// Mitsubishi GX Works2 project: 31-4   PLC: FX3G

// global labels: Global1
VAR_GLOBAL
  start_day AT X007 : BOOL;
  YYYY AT Y007 : BOOL;
  Y1coil AT Y007 : BOOL;
  Reg_WhippedCream AT D1100 : REAL;
END_VAR
VAR_GLOBAL CONSTANT
  constant1_Inventory : REAL := 300;
END_VAR
VAR_GLOBAL
  M_InventoryWhippedCream AT M20 : BOOL;
  Reg_Biscwit AT D1102 : REAL;
END_VAR
VAR_GLOBAL CONSTANT
  constant2_Inventory : REAL := 6;
END_VAR
VAR_GLOBAL
  M_InventoryBiscwit AT Y007 : BOOL;
  Reg_Chochlet AT D1104 : REAL;
END_VAR
VAR_GLOBAL CONSTANT
  constant3_Inventory : REAL := 300;
END_VAR
VAR_GLOBAL
  M_InventoryChochlet AT Y007 : BOOL;
  M_InvetoryWhippedCream AT M20 : BOOL;
  M_InvetoryBiscwit AT M21 : BOOL;
  M_InvetoryChochlet AT M22 : BOOL;
  M_canStartDay AT M0 : BOOL;
  M_toStart AT M1 : BOOL;
  M_InvetoryWhippedCream1 AT M20 : BOOL;
  M_InvetoryBiscwit1 AT M21 : BOOL;
  M_InvetoryChochlet1 AT M22 : BOOL;
  TEXT AT Y011 : BOOL;
  TC_CloseDayTimer_3 AT TC3 : BOOL;
END_VAR
VAR_GLOBAL CONSTANT
  CONSTANT30_word : INT := 30;
END_VAR
VAR_GLOBAL
  lamp1 AT TS1 : BOOL;
  M_stoptDay AT M0 : BOOL;
  tozilof AT X011 : BOOL;
  M_foundMinimum AT X011 : BOOL;
  X011ToStart AT X011 : BOOL;
END_VAR
VAR_GLOBAL CONSTANT
  REG_MinimumCream : REAL := 300;
END_VAR
VAR_GLOBAL
  Reg_sprinkling AT D1106 : REAL;
  M007t AT M7 : BOOL;
  check7 AT M7 : BOOL;
END_VAR
VAR_GLOBAL CONSTANT
  constant1_WhippedCream : REAL := 300;
  constant_WhippedCream : REAL := 300;
  constant_Biscwit : REAL := 6;
  constant_Chochlet : REAL := 240;
  T300Cream : REAL := 300;
  CONSTANT0_float : REAL := 700;
  CONSTANT_CHOCHOLET : REAL := 500;
  CONSTANT_WP : REAL := 300;
  CONSTANT_CH : REAL := 500;
  CONSTANT_BI : REAL := 100;
END_VAR
VAR_GLOBAL
  Reset_Inventory AT M2 : BOOL;
  lamp0 AT M3 : BOOL;
  lamp00 AT M3 : BOOL;
  light0 AT M81 : BOOL;
  light1 AT M82 : BOOL;
  lamp01 AT M3 : BOOL;
END_VAR
VAR_GLOBAL CONSTANT
  TV20 : INT := 5;
END_VAR
VAR_GLOBAL
  TC_light_1 AT TC1 : BOOL;
  TS_light_0 AT TS0 : BOOL;
  TC_light_0 AT TC0 : BOOL;
  TS_light_1 AT TS1 : BOOL;
  start_dipping AT X006 : BOOL;
  SW_AnalogInput1 AT D8280 : INT;
  M_dipping AT M4 : BOOL;
END_VAR
VAR_GLOBAL CONSTANT
  CONSTANT382_1inanalog : INT := 382;
END_VAR
VAR_GLOBAL
  M_CheckDipping AT M5 : BOOL;
END_VAR
VAR_GLOBAL CONSTANT
  CONSTANT2020_5inanalog : INT := 2020;
END_VAR
VAR_GLOBAL
  M_CheckDipping5 AT M6 : BOOL;
  M_CheckDipping1 AT M5 : BOOL;
  lamp3 AT M8 : BOOL;
  SenTouch AT X001 : BOOL;
  Camera AT X002 : BOOL;
  EmergencyButton AT X005 : BOOL;
  SenTemp30 AT X003 : BOOL;
  SenTemp15 AT X004 : BOOL;
  OpenSprinkling AT M33 : BOOL;
  StartSprinkling AT X010 : BOOL;
  OpenSprinkling1 AT M6 : BOOL;
  SprinklingIsOpen AT Y004 : BOOL;
END_VAR
VAR_GLOBAL CONSTANT
  CONSTANT0_1inanalog : INT;
  CONSTANT1995_5inanalog : INT := 1995;
  CONSTANT0_0inanalog : INT;
  CONSTANT3999_10inanalog : INT := 3999;
END_VAR
VAR_GLOBAL
  M_CheckDipping2 AT M55 : BOOL;
END_VAR
VAR_GLOBAL CONSTANT
  CONSTANT2389_6inanalog : INT := 2389;
END_VAR
VAR_GLOBAL
  M_CheckDipping3 AT M66 : BOOL;
END_VAR
VAR_GLOBAL CONSTANT
  CONSTANT_CHOCHOLET20 : REAL := 120;
  CONSTANT_CHOCHOLET40 : REAL := 240;
END_VAR
VAR_GLOBAL
  YY00 AT Y000 : BOOL;
  YY11 AT Y001 : BOOL;
  Reg_dippingToDelte AT D1110 : INT;
  Reg_dipping AT D1112 : REAL;
  Dipping20On AT M11 : BOOL;
  Dipping40On AT M12 : BOOL;
  TC4 AT TC4 : BOOL;
  TC_QA_TEST_PASSED AT TC4 : BOOL;
  TC_4 AT TC4 : BOOL;
END_VAR
VAR_GLOBAL CONSTANT
  CONSTANT50 : INT := 50;
END_VAR
VAR_GLOBAL
  TS_4 AT TS4 : BOOL;
  y_3 AT Y003 : BOOL;
END_VAR
VAR_GLOBAL CONSTANT
  CONSTANT500 : INT := 50;
END_VAR
VAR_GLOBAL
  Start_packing AT X000 : BOOL;
END_VAR
VAR_GLOBAL CONSTANT
  Constant5 : INT := 5;
END_VAR
VAR_GLOBAL
  CC_Start_Squeeze_0 AT CC0 : BOOL;
  CC_counting_0 AT CC0 : BOOL;
  CS0_COUNTING AT CS0 : BOOL;
  Y2_ON AT Y002 : BOOL;
END_VAR
VAR_GLOBAL CONSTANT
  Constant6 : INT := 6;
END_VAR
VAR_GLOBAL
  CS1_COUNTING AT CS1 : BOOL;
  CC_counting_1 AT CC1 : BOOL;
END_VAR
VAR_GLOBAL CONSTANT
  CONSTANT_1 : REAL := 6;
  CONSTANT_6 : REAL := 6;
END_VAR
VAR_GLOBAL
  addto8282 AT D8282 : INT;
END_VAR
VAR_GLOBAL CONSTANT
  CONSTANT_10 : REAL := 10;
END_VAR
VAR_GLOBAL
  CS_counting_0 AT CS0 : BOOL;
  CS_counting_1 AT CS1 : BOOL;
  check_sprinkling AT M77 : BOOL;
  TC_total AT TC4 : BOOL;
END_VAR
VAR_GLOBAL CONSTANT
  TV40 : INT := 40;
END_VAR
VAR_GLOBAL
  M_300 AT M300 : BOOL;
  TS_total AT TS4 : BOOL;
  Ymove0 AT Y000 : BOOL;
  Ymove1 AT Y001 : BOOL;
  Step1 AT M101 : BOOL;
  Step2 AT M102 : BOOL;
  Step3 AT M103 : BOOL;
  Step4 AT M104 : BOOL;
  StepFinal AT M100 : BOOL;
  TC_5 AT TC5 : BOOL;
  TS_5 AT TS5 : BOOL;
  ToStep2 AT M102 : BOOL;
  TS_CloseDayTimer_3 AT TS3 : BOOL;
  Ym11 AT Y011 : BOOL;
  Step4M AT M444 : BOOL;
  Step5 AT M105 : BOOL;
  Step3M AT M333 : BOOL;
  Reg_Count_to8282 AT D1116 : INT;
  Reg_Countt AT D1122 : REAL;
  mtototot99 AT M99 : BOOL;
  Reg_Countt10 AT D1124 : REAL;
END_VAR
VAR_GLOBAL CONSTANT
  COcococo23 : INT := 2;
  CON400 : INT := 400;
  CON40 : REAL := 40;
END_VAR
VAR_GLOBAL
  Dippingn AT M11 : BOOL;
  goagain AT M110 : BOOL;
  X_11 AT Y011 : BOOL;
  Reg_fill_WP AT D1130 : REAL;
  Reg_fill_CH AT D1132 : REAL;
  Reg_fill_BI AT D1134 : REAL;
  M_reset AT M64 : BOOL;
  M_step1 AT M63 : BOOL;
END_VAR

// task Task_01 (event TRUE, interval 0, priority 31): POU_01

PROGRAM POU_01
(* structured ladder/FBD written out as ST: instructions are called as NAME(EN, inputs, outputs); _pN, _eN, _tN stand for wires *)
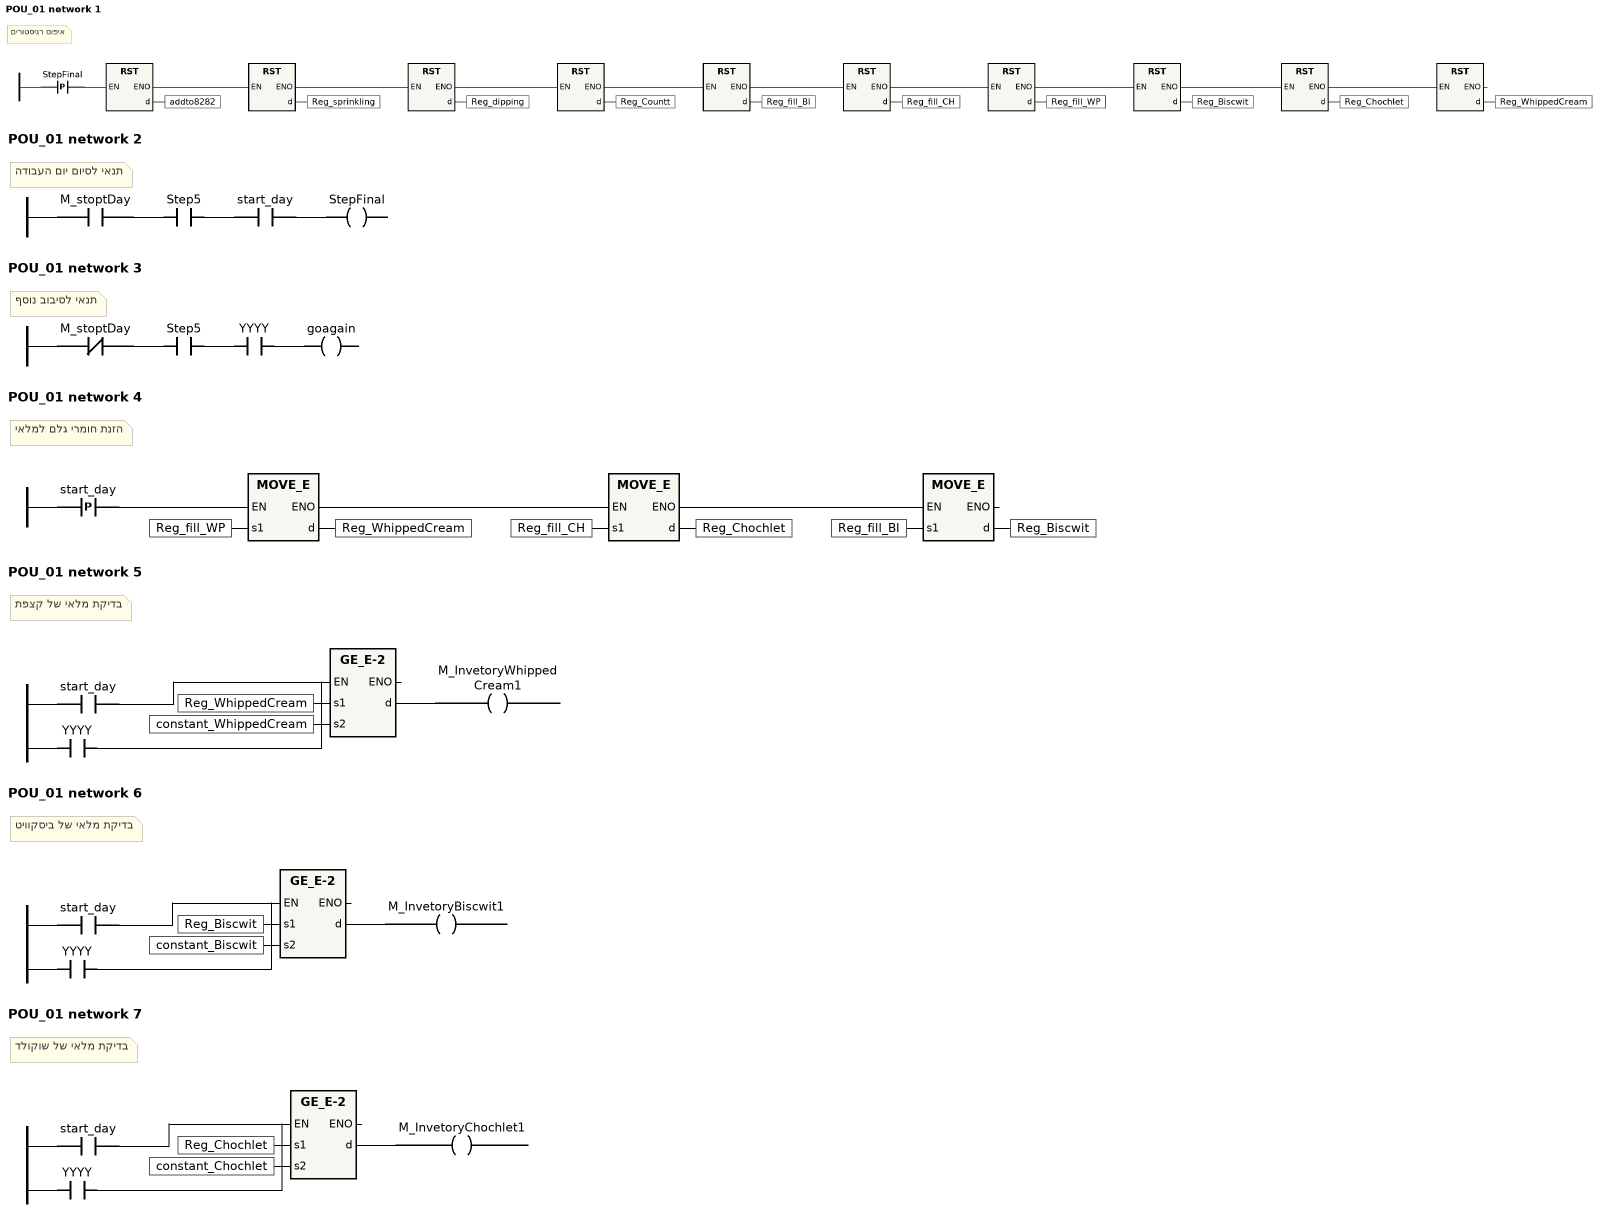
(* network 1 *)
(* איפוס רגיסטורים *)
_e1 := RST(LDP(TRUE, StepFinal), addto8282);
_e2 := RST(_e1, Reg_sprinkling);
_e3 := RST(_e2, Reg_dipping);
_e4 := RST(_e3, Reg_Countt);
_e5 := RST(_e4, Reg_fill_BI);
_e6 := RST(_e5, Reg_fill_CH);
_e7 := RST(_e6, Reg_fill_WP);
_e8 := RST(_e7, Reg_Biscwit);
_e9 := RST(_e8, Reg_Chochlet);
RST(_e9, Reg_WhippedCream);
(* network 2 *)
(* תנאי לסיום יום העבודה *)
StepFinal := M_stoptDay AND Step5 AND start_day;
(* network 3 *)
(* תנאי לסיבוב נוסף *)
goagain := NOT M_stoptDay AND Step5 AND YYYY;
(* network 4 *)
(* הזנת חומרי גלם למלאי *)
_e1 := MOVE_E(LDP(TRUE, start_day), Reg_fill_WP, Reg_WhippedCream);
_e2 := MOVE_E(_e1, Reg_fill_CH, Reg_Chochlet);
MOVE_E(_e2, Reg_fill_BI, Reg_Biscwit);
(* network 5 *)
(* בדיקת מלאי של קצפת *)
GE_E(start_day OR YYYY, Reg_WhippedCream, constant_WhippedCream, _t1);
M_InvetoryWhippedCream1 := _t1;
(* network 6 *)
(* בדיקת מלאי של ביסקוויט *)
GE_E(start_day OR YYYY, Reg_Biscwit, constant_Biscwit, _t1);
M_InvetoryBiscwit1 := _t1;
(* network 7 *)
(* בדיקת מלאי של שוקולד *)
GE_E(start_day OR YYYY, Reg_Chochlet, constant_Chochlet, _t1);
M_InvetoryChochlet1 := _t1;
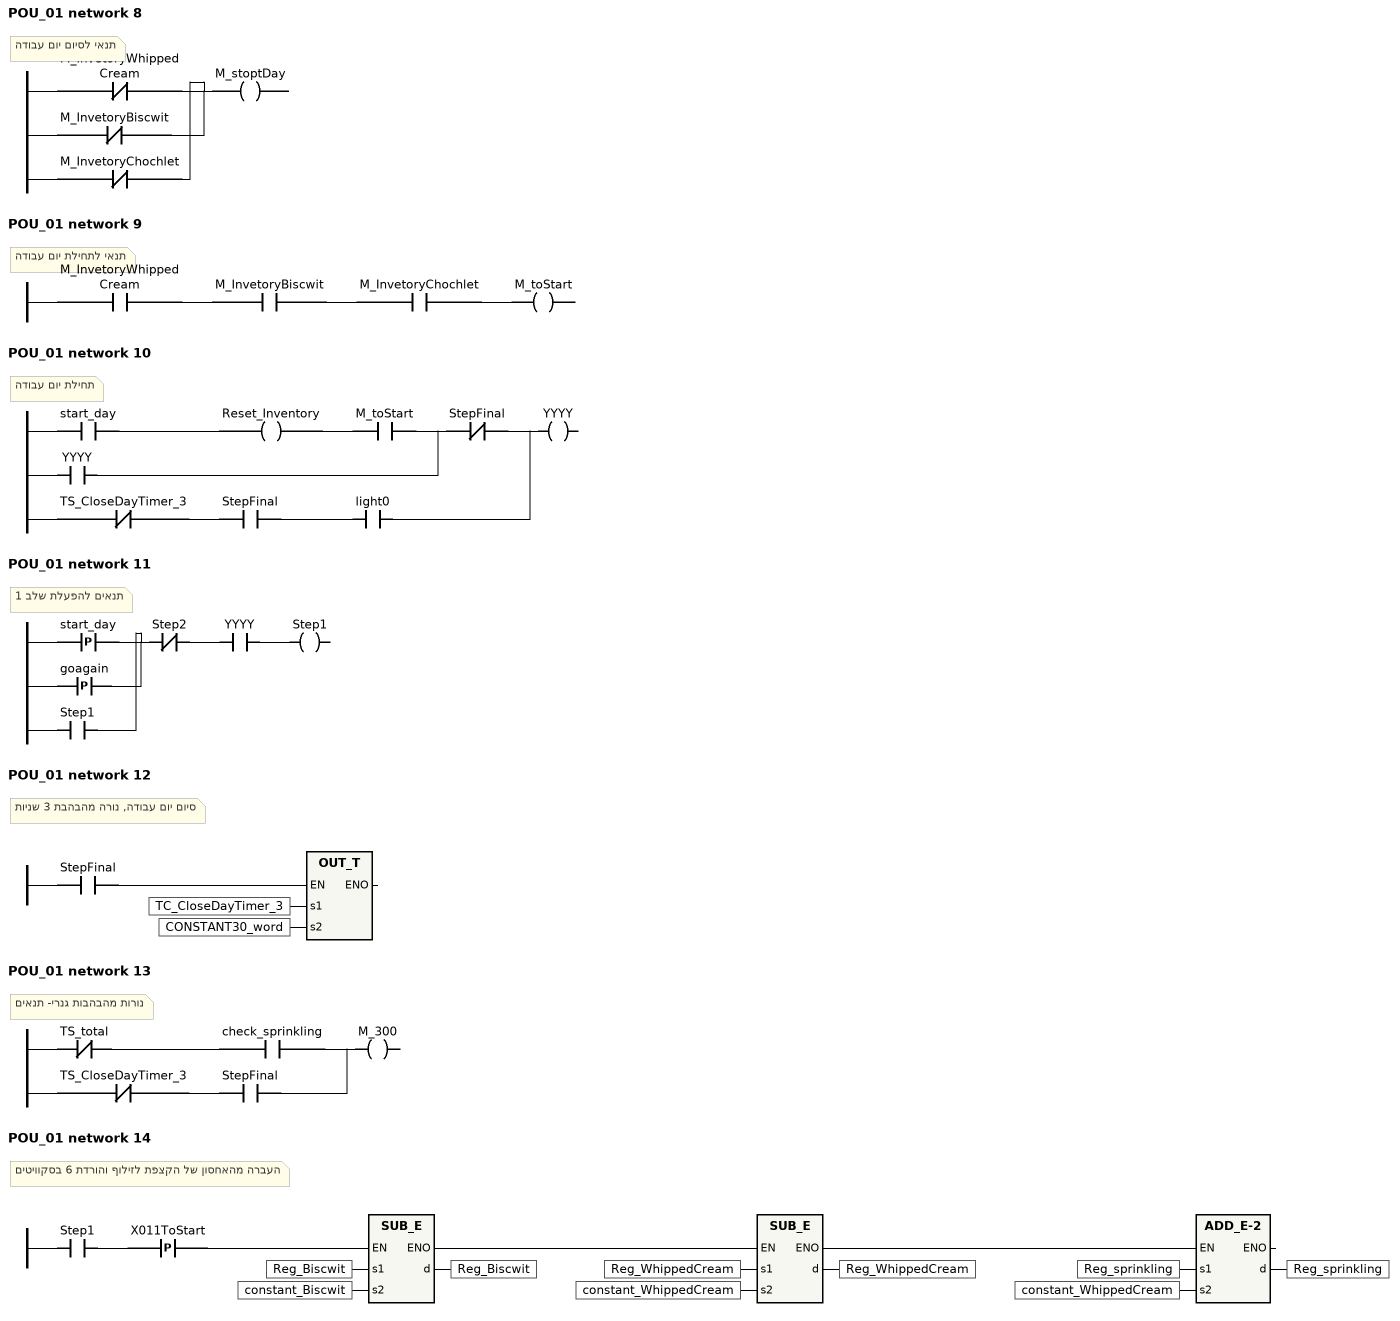
(* network 8 *)
(* תנאי לסיום יום עבודה *)
M_stoptDay := (NOT M_InvetoryWhippedCream) OR (NOT M_InvetoryBiscwit) OR (NOT M_InvetoryChochlet);
(* network 9 *)
(* תנאי לתחילת יום עבודה *)
M_toStart := M_InvetoryWhippedCream AND M_InvetoryBiscwit AND M_InvetoryChochlet;
(* network 10 *)
(* תחילת יום עבודה *)
Reset_Inventory := start_day;
YYYY := (((start_day AND M_toStart) OR YYYY) AND NOT StepFinal) OR (NOT TS_CloseDayTimer_3 AND StepFinal AND light0);
(* network 11 *)
(* תנאים להפעלת שלב 1 *)
Step1 := ((LDP(TRUE, start_day) OR LDP(TRUE, goagain) OR Step1) AND NOT Step2) AND YYYY;
(* network 12 *)
(* סיום יום עבודה, נורה מהבהבת 3 שניות *)
OUT_T(StepFinal, TC_CloseDayTimer_3, CONSTANT30_word);
(* network 13 *)
(* נורות מהבהבות גנרי- תנאים *)
M_300 := (NOT TS_total AND check_sprinkling) OR (NOT TS_CloseDayTimer_3 AND StepFinal);
(* network 14 *)
(* העברה מהאחסון של הקצפת לזילוף והורדת 6 בסקוויטים *)
_e1 := SUB_E(Step1 AND LDP(TRUE, X011ToStart), Reg_Biscwit, constant_Biscwit, Reg_Biscwit);
_e2 := SUB_E(_e1, Reg_WhippedCream, constant_WhippedCream, Reg_WhippedCream);
ADD_E(_e2, Reg_sprinkling, constant_WhippedCream, Reg_sprinkling);
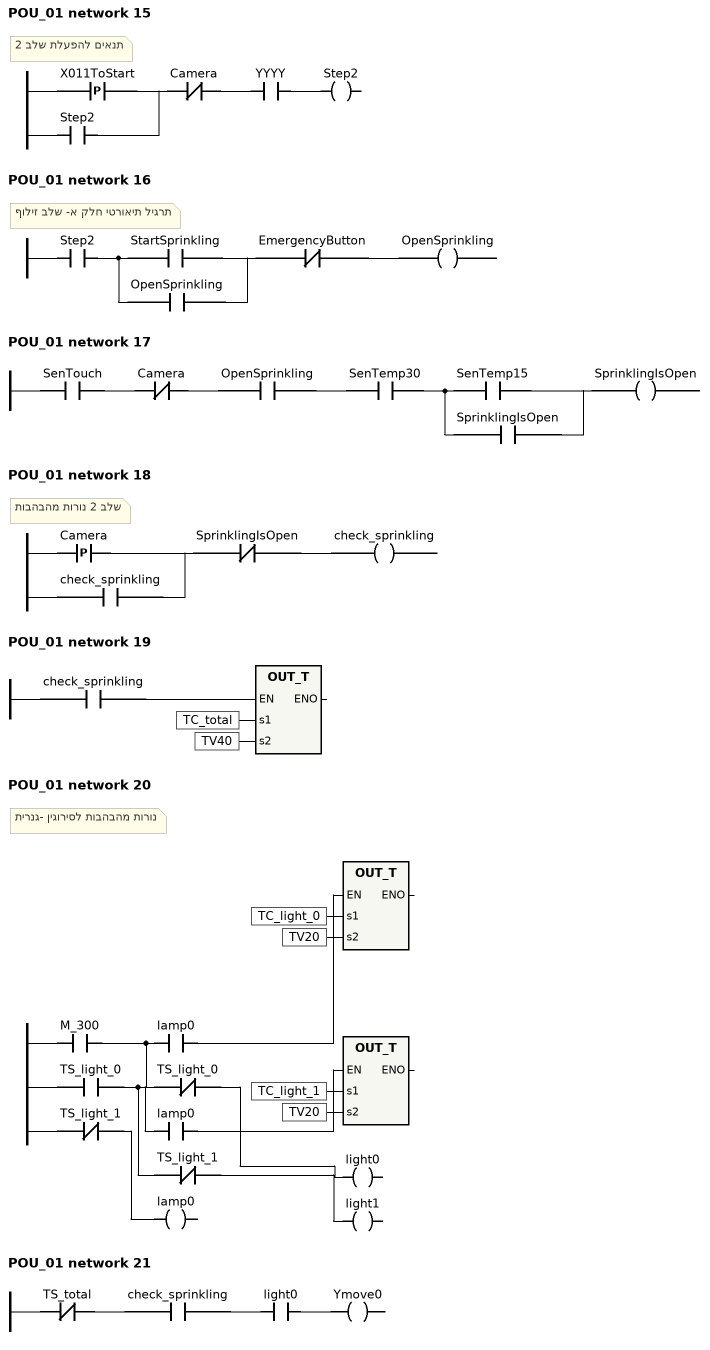
(* network 15 *)
(* תנאים להפעלת שלב 2 *)
Step2 := ((LDP(TRUE, X011ToStart) OR Step2) AND NOT Camera) AND YYYY;
(* network 16 *)
(* תרגיל תיאורטי חלק א- שלב זילוף *)
OpenSprinkling := ((Step2 AND StartSprinkling) OR (Step2 AND OpenSprinkling)) AND NOT EmergencyButton;
(* network 17 *)
_p1 := SenTouch AND NOT Camera AND OpenSprinkling AND SenTemp30;
SprinklingIsOpen := (_p1 AND SenTemp15) OR (_p1 AND SprinklingIsOpen);
(* network 18 *)
(* שלב 2 נורות מהבהבות *)
check_sprinkling := (LDP(TRUE, Camera) OR check_sprinkling) AND NOT SprinklingIsOpen;
(* network 19 *)
OUT_T(check_sprinkling, TC_total, TV40);
(* network 20 *)
(* נורות מהבהבות לסירוגין -גנרית *)
OUT_T(M_300 AND lamp0, TC_light_0, TV20);
light0 := M_300 AND NOT TS_light_0;
OUT_T(TS_light_0 AND lamp0, TC_light_1, TV20);
light1 := TS_light_0 AND NOT TS_light_1;
lamp0 := NOT TS_light_1;
(* network 21 *)
Ymove0 := NOT TS_total AND check_sprinkling AND light0;
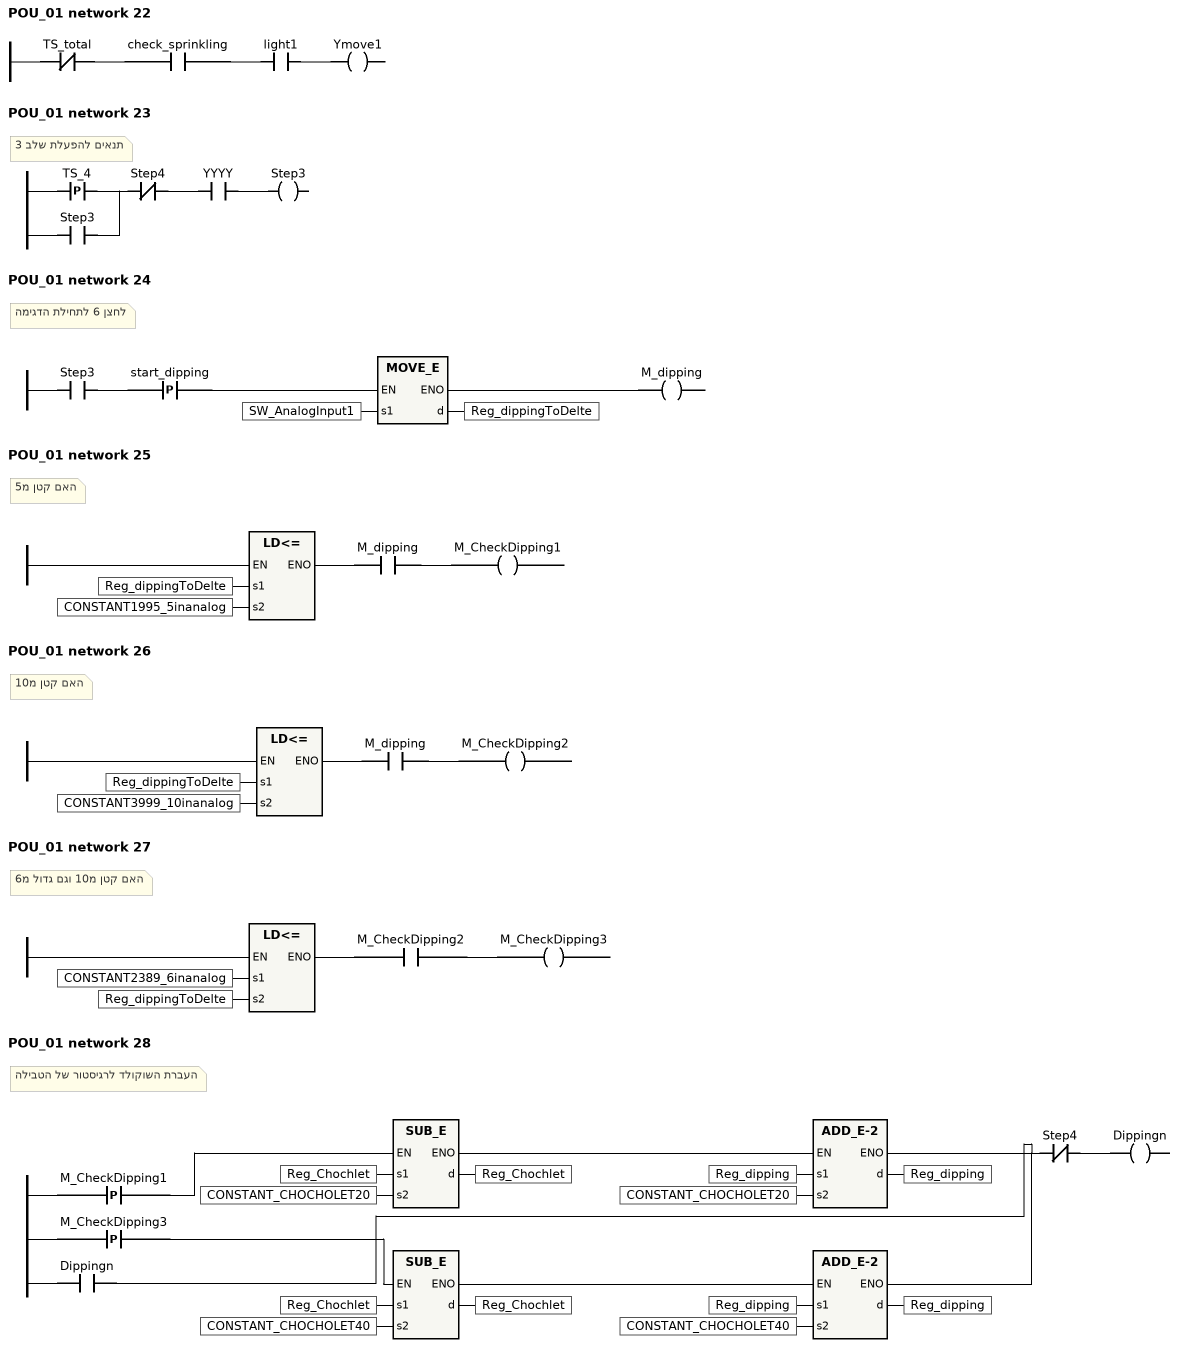
(* network 22 *)
Ymove1 := NOT TS_total AND check_sprinkling AND light1;
(* network 23 *)
(* תנאים להפעלת שלב 3 *)
Step3 := ((LDP(TRUE, TS_4) OR Step3) AND NOT Step4) AND YYYY;
(* network 24 *)
(* לחצן 6 לתחילת הדגימה *)
_e1 := MOVE_E(Step3 AND LDP(TRUE, start_dipping), SW_AnalogInput1, Reg_dippingToDelte);
M_dipping := _e1;
(* network 25 *)
(* האם קטן מ5 *)
_e1 := LD<=(TRUE, Reg_dippingToDelte, CONSTANT1995_5inanalog);
M_CheckDipping1 := _e1 AND M_dipping;
(* network 26 *)
(* האם קטן מ10 *)
_e1 := LD<=(TRUE, Reg_dippingToDelte, CONSTANT3999_10inanalog);
M_CheckDipping2 := _e1 AND M_dipping;
(* network 27 *)
(* האם קטן מ10 וגם גדול מ6 *)
_e1 := LD<=(TRUE, CONSTANT2389_6inanalog, Reg_dippingToDelte);
M_CheckDipping3 := _e1 AND M_CheckDipping2;
(* network 28 *)
(* העברת השוקולד לרגיסטור של הטבילה *)
_e1 := SUB_E(LDP(TRUE, M_CheckDipping1), Reg_Chochlet, CONSTANT_CHOCHOLET20, Reg_Chochlet);
_e2 := ADD_E(_e1, Reg_dipping, CONSTANT_CHOCHOLET20, Reg_dipping);
_e3 := SUB_E(LDP(TRUE, M_CheckDipping3), Reg_Chochlet, CONSTANT_CHOCHOLET40, Reg_Chochlet);
_e4 := ADD_E(_e3, Reg_dipping, CONSTANT_CHOCHOLET40, Reg_dipping);
Dippingn := (_e2 OR _e4 OR Dippingn) AND NOT Step4;
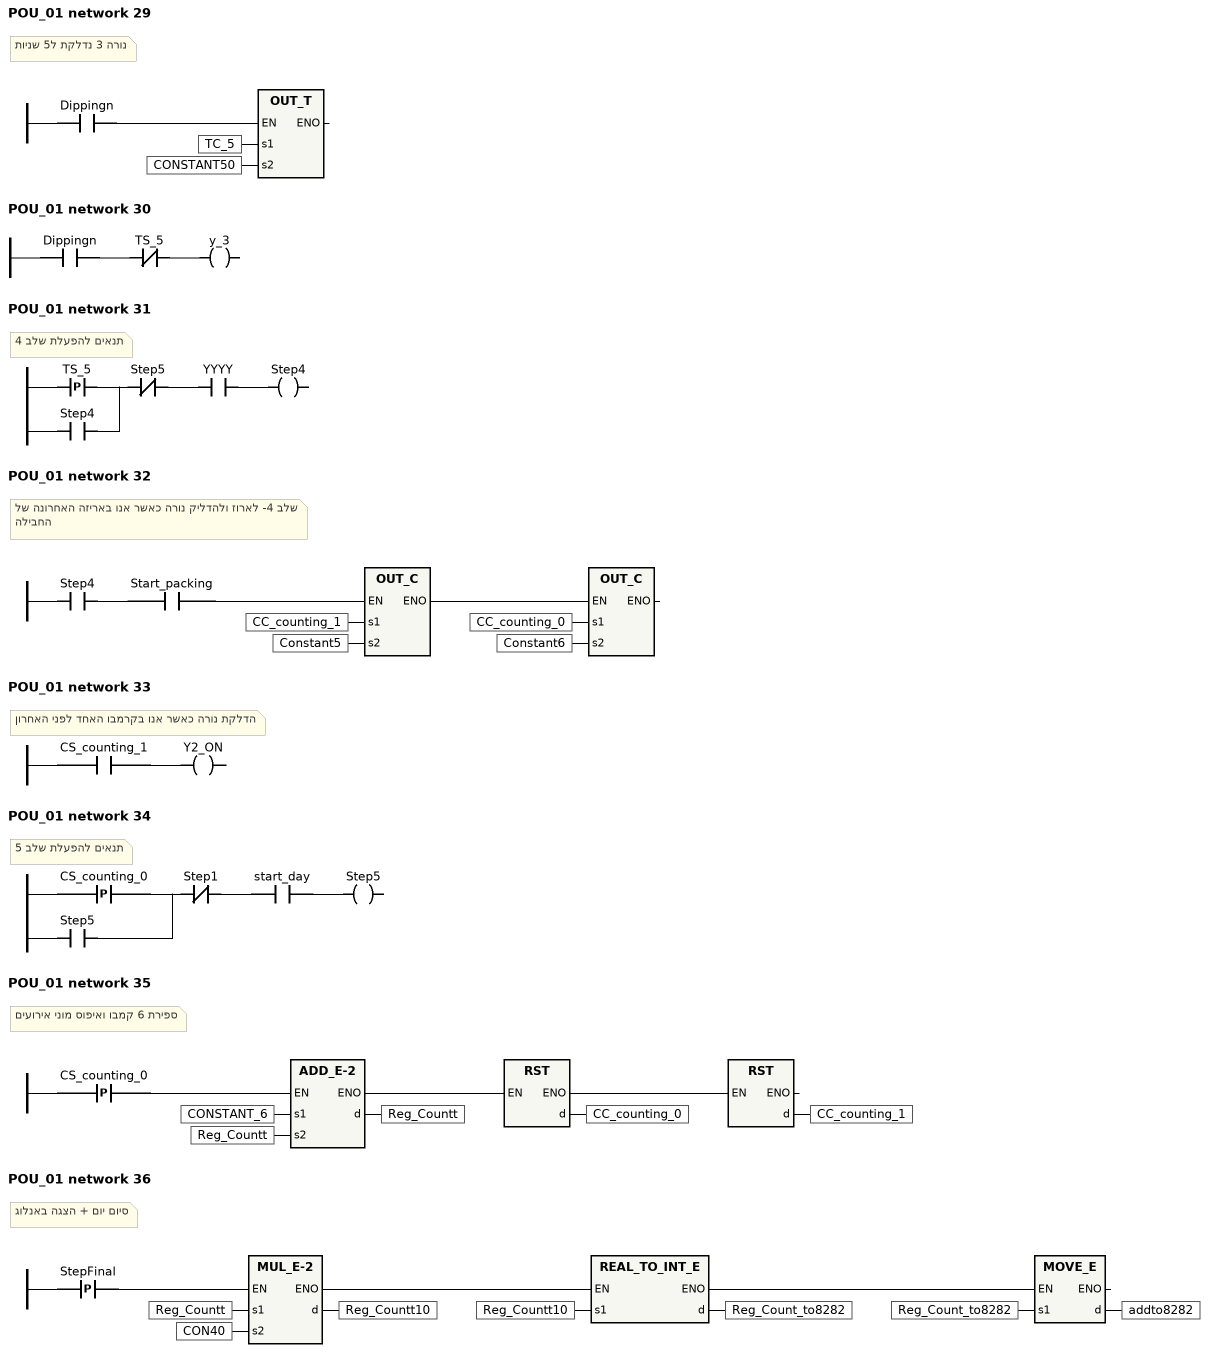
(* network 29 *)
(* נורה 3 נדלקת ל5 שניות *)
OUT_T(Dippingn, TC_5, CONSTANT50);
(* network 30 *)
y_3 := Dippingn AND NOT TS_5;
(* network 31 *)
(* תנאים להפעלת שלב 4 *)
Step4 := ((LDP(TRUE, TS_5) OR Step4) AND NOT Step5) AND YYYY;
(* network 32 *)
(* שלב 4- לארוז ולהדליק נורה כאשר אנו באריזה האחרונה של החבילה *)
_e1 := OUT_C(Step4 AND Start_packing, CC_counting_1, Constant5);
OUT_C(_e1, CC_counting_0, Constant6);
(* network 33 *)
(* הדלקת נורה כאשר אנו בקרמבו האחד לפני האחרון *)
Y2_ON := CS_counting_1;
(* network 34 *)
(* תנאים להפעלת שלב 5 *)
Step5 := ((LDP(TRUE, CS_counting_0) OR Step5) AND NOT Step1) AND start_day;
(* network 35 *)
(* ספירת 6 קמבו ואיפוס מוני אירועים *)
_e1 := ADD_E(LDP(TRUE, CS_counting_0), CONSTANT_6, Reg_Countt, Reg_Countt);
_e2 := RST(_e1, CC_counting_0);
RST(_e2, CC_counting_1);
(* network 36 *)
(* סיום יום + הצגה באנלוג *)
_e1 := MUL_E(LDP(TRUE, StepFinal), Reg_Countt, CON40, Reg_Countt10);
_e2 := REAL_TO_INT_E(_e1, Reg_Countt10, Reg_Count_to8282);
MOVE_E(_e2, Reg_Count_to8282, addto8282);
END_PROGRAM
